(*
SPDX-FileCopyrightText: © 2026 Oleksandr Tiutyk <trofimich@gmail.com>
SPDX-License-Identifier: MIT
License: https://opensource.org/license/mit
*)

{attribute 'no_explicit_call' := 'do not call this function block directly'} 
FUNCTION_BLOCK WideStringSplittingEnumerator EXTENDS Object IMPLEMENTS IEnumerator
VAR_OUTPUT
	SourceString : POINTER TO WSTRING;
	SourceStringLength : UDINT;
	SourceStringSize : UDINT;
	Separator : WSTRING;
	SeparatorLength : UDINT;
	MaxCount : UDINT := 0;
	TrimEntries : BOOL := FALSE;
	RemoveEmptyEntries : BOOL := FALSE;	
END_VAR
VAR
	{attribute 'hide'} 
	_ClassName : STRING := __POUNAME();

	{attribute 'hide'} 
	_CurrentString : POINTER TO WSTRING;
	{attribute 'hide'} 
	_CurrentStringLength : UDINT;
	{attribute 'hide'} 
	_CurrentEntry : POINTER TO WSTRING;
	{attribute 'hide'} 
	_CurrentEntrySize : UDINT;
	{attribute 'hide'} 
	_EntryCount : UDINT; 
END_VAR

{attribute 'monitoring' := 'call'}
PROPERTY ClassName : REFERENCE TO STRING
GET
ClassName REF= _ClassName;
END_GET
END_PROPERTY

(*!
<summary>Shows curent collection element</summary>
*)

{attribute 'monitoring' := 'call'}
PROPERTY Current : REFERENCE TO GENERIC_VALUE
GET
VAR_INST
	genericValue : GENERIC_VALUE;
END_VAR
IF _CurrentEntry <> 0 AND_THEN _CurrentEntrySize > 0 THEN
	genericValue := GenericValueFactory.FromParts(GENERIC_TYPE_CLASS.STRING_UTF16, _CurrentEntry, _CurrentEntrySize, GENERIC_MEMORY_MANAGEMENT_BEHAVIOR.STORE_ORIGINAL_REFERENCE_AND_NOT_OWNS_MEMORY);
ELSE
	genericValue.Reset();
END_IF

Current REF= genericValue;
END_GET
END_PROPERTY

PROPERTY CurrentEntry : REFERENCE TO WSTRING
GET
IF _CurrentEntry <> 0 THEN
	CurrentEntry REF= _CurrentEntry^;	
END_IF
END_GET
END_PROPERTY

//!<param name="bInCopyCode">if TRUE, the exit method is called for exiting an instance that is copied afterwards (online change).</param>

METHOD FB_exit : BOOL
VAR_INPUT
	
	bInCopyCode	: BOOL;
END_VAR
IF _CurrentEntry <> 0 THEN
	__DELETE(_CurrentEntry);
END_IF
END_METHOD

METHOD INTERNAL Initialize
VAR_INPUT
	sourceString : POINTER TO WSTRING;
	separator : WSTRING;
	maxCount : UDINT;
	trimEntries : BOOL;
	removeEmptyEntries : BOOL;
END_VAR
THIS^.SourceString := sourceString;
THIS^.SourceStringLength := WideStrings.InternalGetLength(sourceString);
THIS^.SourceStringSize := THIS^.SourceStringLength + WideStrings.CharSize; 
THIS^.Separator := separator;
THIS^.SeparatorLength := WideStrings.InternalGetLength(ADR(separator));
THIS^.MaxCount := maxCount;
THIS^.TrimEntries := trimEntries;
THIS^.RemoveEmptyEntries := removeEmptyEntries;

_CurrentString := THIS^.SourceString;

Reset();
END_METHOD

METHOD MoveNext : BOOL
VAR
	separatorPosition : UDINT;
END_VAR
START:

IF _CurrentEntry <> 0 THEN
	_CurrentEntrySize := 0;
	
	__DELETE(_CurrentEntry);
END_IF

IF _CurrentString = 0 OR_ELSE _CurrentStringLength = 0 OR_ELSE Separator = "" OR_ELSE (MaxCount > 0 AND_THEN _EntryCount >= MaxCount) THEN
	RETURN;
END_IF

IF WideStrings.InternalFind(_CurrentString, _CurrentStringLength, ADR(Separator), SeparatorLength, position => separatorPosition) THEN
	_CurrentEntrySize := separatorPosition * WideStrings.CharSize;
	_CurrentEntry := __NEW(BYTE, _CurrentEntrySize);

	Tc2_System.MEMCPY(_CurrentEntry, _CurrentString, (separatorPosition - 1) * WideStrings.CharSize);
	Tc2_System.MEMSET(_CurrentEntry + ((separatorPosition - 1) * WideStrings.CharSize), 0, WideStrings.CharSize);

	_CurrentString := _CurrentString + ((separatorPosition - 1) * WideStrings.CharSize) + (SeparatorLength * WideStrings.CharSize);
	_CurrentStringLength := _CurrentStringLength - separatorPosition + 1 - SeparatorLength;
ELSE	
	_CurrentEntrySize := _CurrentStringLength + WideStrings.CharSize;	
	_CurrentEntry := __NEW(BYTE, _CurrentEntrySize);
	
	Tc2_System.MEMCPY(_CurrentEntry, _CurrentString, _CurrentStringLength + WideStrings.CharSize);
	
	_CurrentString := 0;
	_CurrentStringLength := 0;
END_IF

IF TrimEntries THEN
	WideStrings.TrimChar(_CurrentEntry^);
END_IF

IF RemoveEmptyEntries AND_THEN _CurrentEntry^ = "" THEN
	JMP START;
END_IF

_EntryCount := _EntryCount + 1;

MoveNext := TRUE;
END_METHOD

{attribute 'monitoring' := 'call'}
PROPERTY NamespaceName : REFERENCE TO STRING
GET
NamespaceName REF= CurrentNamespace.Name;
END_GET
END_PROPERTY

(*!
<summary>Releases the current fragment and resets iteration to before the first entry.</summary>
<description>
Preserves splitting settings and does not allocate memory or modify the source string.
Previously borrowed fragment addresses and references become invalid.
The initialized source string must remain alive and unchanged throughout iteration.
Repeated Reset calls are allowed, including before iteration and after its end.
</description>
*)
METHOD Reset
IF _CurrentEntry <> 0 THEN
	__DELETE(_CurrentEntry);
END_IF

_CurrentEntry := 0;
_CurrentEntrySize := 0;

_CurrentString := SourceString;
_CurrentStringLength := SourceStringLength;
_EntryCount := 0;
END_METHOD

{attribute 'monitoring' := 'call'}
PROPERTY SelfSize : ULINT
GET
SelfSize := XSIZEOF(THIS^);
END_GET
END_PROPERTY

END_FUNCTION_BLOCK

(* stored: Version 1.1.0.1
   POU WideStringSplittingEnumerator: Id {cd3c3f30-cd38-4659-b9c4-859e877b4baf}, SpecialFunc None
   Property ClassName: Id {eb782797-fea3-47ac-a8db-cbfc72d737be}
   Get Get: Id {b0de37f0-477e-4092-a2e4-1e3cd48b7e08}
   Property Current: Id {a33a22ac-5669-4623-936f-19fdd6a797a9}
   Get Get: Id {b343fd78-0841-4c7a-bd2d-6b447815e0a9}
   Property CurrentEntry: Id {f4b2ce05-56f1-4a2a-ab8a-2d63ad7de743}
   Get Get: Id {859e54d6-429d-47fd-a753-3e8e965a0bc3}
   Method FB_exit: Id {d23faa7c-5379-472c-b75f-ff9aa468fe1d}
   Method Initialize: Id {efd8c83e-84af-4552-92cf-49864ca5b37a}
   Method MoveNext: Id {6f4c66bb-70e6-443d-b741-5ac7aedc0a0c}
   Property NamespaceName: Id {606a15c2-aeca-432d-8e3c-a9852072d07e}
   Get Get: Id {8d26a153-dac4-4ce7-b323-94027a2445d2}
   Method Reset: Id {6ff5f895-f51d-4f1c-b79b-00ce34e370cc}
   Property SelfSize: Id {e6e7cb18-6bbe-4fa5-8b86-e60c4005ed50}
   Get Get: Id {6cd74453-76de-45a9-9aff-7d3ec88a250f} *)
